// TwinCAT 3 PLC project Log_Test_Controller
// ProgramVersion: 3.1.4024.0
// libraries:
//   Tc2_Standard, * (Beckhoff Automation GmbH)
//   Tc2_System, * (Beckhoff Automation GmbH)
//   Tc2_Utilities, * (Beckhoff Automation GmbH)
//   Tc3_IotBase, * (Beckhoff Automation GmbH)
//   Tc3_Module, * (Beckhoff Automation GmbH)
//   Tc2_ModbusRTU,3.5.6.0,Beckhoff Automation GmbH
// project tree:
//   DUTs/ ST_PowerMeter.TcDUT
//   GVLs/ GVL.TcGVL
//   / PlcTask.TcTTO
//   POUs/ MAIN.TcPOU, ModbusRTU.TcPOU, MQTT.TcPOU
// real-time tasks:
//   TASK PlcTask: cycle T#10ms, priority 20, ADS port 350
// I/O:
//   DEVICE Device 1 (EtherCAT), AmsNetId 10.200.124.203.2.1
//     Term 1 (EK1200) [EK1200-7000 EtherCAT Power supply (1,5A E-Bus)]
//       Term 2 (EL6021) [EL6021 Interface (RS422/485)]
//       Term 3 (EL9011) [EL9011 End Terminal]
//   DEVICE Device 3 (CX7000), AmsNetId 10.200.124.203.4.1
//   DEVICE Device 5 (COM Port)
// variable links:
//   Log_Test_Controller/Log_Test_Controller Instance <-> Device 1 (EtherCAT)/Term 1 (EK1200)/Term 2 (EL6021)
//     PlcTask Inputs/ModbusRTU.fbEpcMb.InData/D <-> COM TxPDO-Map Inputs/Data In 0
//     PlcTask Inputs/ModbusRTU.fbEpcMb.InData/D @bit {8..168 step 8} <-> COM TxPDO-Map Inputs/Data In {1..21}  (21 links)
//     PlcTask Inputs/ModbusRTU.fbEpcMb.InData/Status <-> COM TxPDO-Map Inputs/Status
//     PlcTask Outputs/ModbusRTU.fbEpcMb.OutData/Ctrl <-> COM RxPDO-Map Outputs/Ctrl
//     PlcTask Outputs/ModbusRTU.fbEpcMb.OutData/D <-> COM RxPDO-Map Outputs/Data Out 0
//     PlcTask Outputs/ModbusRTU.fbEpcMb.OutData/D @bit {8..168 step 8} <-> COM RxPDO-Map Outputs/Data Out {1..21}  (21 links)

CONFIGURATION Log_Test_Controller
    RESOURCE PLC ON TwinCAT3
        TASK PlcTask(INTERVAL := T#10ms, PRIORITY := 20);
        PROGRAM MAIN WITH PlcTask : MAIN;
    END_RESOURCE
END_CONFIGURATION

// ---- DUTs/ST_PowerMeter.TcDUT
TYPE ST_PowerMeter :
STRUCT
	fProp1: WORD;
	fProp2: WORD;
	fProp3: WORD;
	fProp4: WORD;
	fProp5: WORD;
	fProp6: WORD;
	fProp7: WORD;
	fProp8: WORD;
	fProp9: WORD;
	fProp10: WORD;
END_STRUCT
END_TYPE

// ---- GVLs/GVL.TcGVL
{attribute 'qualified_only'}
VAR_GLOBAL
	aMeterData: ARRAY[1..20] OF ST_PowerMeter;
END_VAR

// ---- POUs/MAIN.TcPOU
PROGRAM MAIN
VAR
END_VAR

ModbusRTU();
MQTT();

END_PROGRAM

// ---- POUs/ModbusRTU.TcPOU
PROGRAM ModbusRTU
VAR
	fbEpcMb: ModbusRtuMaster_KL6x22B;
	nMbId: BYTE := 1;
	wQty: WORD := 10;
	wMbAddr: WORD := 20;
	stData: ST_PowerMeter;
	bRead: BOOL;
	fbRTrigRead: R_TRIG;
	nReadState: UINT;
END_VAR

fbRTrigRead(CLK:=bRead, Q=>);

CASE nReadState OF
	0:
		bRead := TRUE;
		IF fbRTrigRead.Q THEN
			nReadState := 1;
		END_IF
	1:
		bRead := FALSE;
		IF NOT fbEpcMb.BUSY AND NOT fbEpcMb.Error THEN
			GVL.aMeterData[nMbId] := stData;
			IF nMbId < 20 THEN
				nMbId := nMbId + 1;
			ELSE
				nMbId := 1;
			END_IF	
			nReadState := 0;
		END_IF
END_CASE

fbEpcMb.ReadRegs(
	UnitID:= nMbId, 
	Quantity:= wQty, 
	MBAddr:= wMbAddr, 
	cbLength:= SIZEOF(stData), 
	pMemoryAddr:= ADR(stData), 
	Execute:= fbRTrigRead.Q, 
	Timeout:= T#2S, 
	BUSY=> , 
	Error=> , 
	ErrorId=> , 
	cbRead=> );

END_PROGRAM

// ---- POUs/MQTT.TcPOU
PROGRAM MQTT
VAR
	fbMqttClient: FB_IotMqttClient;
	bSetParameter: BOOL:=TRUE;
	bConnect: BOOL:= TRUE;
	(* published message *)
    sTopicPub   : STRING(255) := 'LongAn/DucHoa/DuyTan/Station2/Device';
    sPayloadPub : STRING(255):='';
	buffer		: STRING(255):='';
	name: STRING(255):= 'Hoang Minh Tri';
    i : INT:=1;
	nState : INT:=0;
    fbTimer : TON := (PT:=T#0.5S);
    fbMessageQueue : FB_IotMqttMessageQueue;
	fbFormat: FB_FormatString;
END_VAR

		IF bSetParameter THEN
			bSetParameter               := FALSE;
			fbMqttClient.sHostName      := '192.168.1.253';
			fbMqttClient.nHostPort      := 1883;
		//  fbMqttClient.sClientId      := 'MyTcMqttClient'; 
			fbMqttClient.sTopicPrefix   := ''; 
		//  fbMqttClient.nKeepAlive     := 60; 
		//  fbMqttClient.sUserName      := ;
		//  fbMqttClient.sUserPassword  := ; 
		//  fbMqttClient.stWill         := ; 
		//  fbMqttClient.stTLS          := ;
			fbMqttClient.ipMessageQueue := fbMessageQueue;
		END_IF
fbMqttClient.Execute(bConnect);
CASE nState OF
	0: //Connection establishment
		nState:= 10;
	10: // -----------CONCAT STRING FOR payload---------------
		
		fbFormat(
		sFormat:= '%d,%d,%d,%d,%d,%d,%d,%d,%d,%d ',
			arg1:= F_WORD(GVL.aMeterData[i].fProp1),
			arg2:= F_WORD(GVL.aMeterData[i].fProp2),
			arg3:= F_WORD(GVL.aMeterData[i].fProp3),
			arg4:= F_WORD(GVL.aMeterData[i].fProp4),
			arg5:= F_WORD(GVL.aMeterData[i].fProp5),
			arg6:= F_WORD(GVL.aMeterData[i].fProp6),
			arg7:= F_WORD(GVL.aMeterData[i].fProp7),
			arg8:= F_WORD(GVL.aMeterData[i].fProp8),
			arg9:= F_WORD(GVL.aMeterData[i].fProp9),
			arg10:= F_WORD(GVL.aMeterData[i].fProp10),
			bError => ,
			nErrId => ,
			sOut => sPayloadPub
		);
		sTopicPub:= CONCAT(sTopicPub,INT_TO_STRING(i));
		nState:= 20;
	20://-------------------Publish data to broker----------------
		IF fbMqttClient.bConnected THEN
			fbMqttClient.Publish(   sTopic:= sTopicPub, 
									pPayload:= ADR(sPayloadPub), nPayloadSize:= LEN2(ADR(sPayloadPub))+1, 
									eQoS:= TcIotMqttQos.AtMostOnceDelivery, bRetain:= FALSE, bQueue:= FALSE );
			sPayloadPub:='';
			sTopicPub:='LongAn/DucHoa/DuyTan/Station2/Device';
			nState:=30;
		END_IF
	30://-------------------Waiting for publishing----------------
		IF NOT fbMqttClient.bError THEN
			fbTimer(IN:=TRUE);
			IF fbTimer.Q THEN // publish new payload every 5 seconds
        		fbTimer(IN:=FALSE);
				IF i = 20 THEN
					i:=1;
				ELSE
					i:=i+1;
				END_IF
				nState:=10;
			END_IF

		END_IF
END_CASE

END_PROGRAM
